// Reads a string field value from the input.
FUNCTION INTERNAL F_ReadStringInternal : HRESULT
VAR_IN_OUT      
    stCtx : ST_ParseContext;
END_VAR
VAR_INPUT
    stAnyStringOut : T_Any;   
END_VAR
VAR
    nStrLength : UDINT;
END_VAR

F_ReadStringInternal := S_OK;

F_ReadStringInternal := F_ParseLength(stCtx, nLength=> nStrLength);
IF FAILED(F_ReadStringInternal) THEN
    RETURN;
END_IF

F_ReadStringInternal := F_ReadRawString(stCtx, nStrLength, stAnyStringOut);

END_FUNCTION

(* stored: Version 1.1.0.1
   POU F_ReadStringInternal: Id {4706b8e4-8703-4440-a040-6ca18bbb6b15}, SpecialFunc None *)
